IF bLoadTara THEN
	bLoadcell_fbcmd	:= LoadCell.GetTara();
END_IF
tmrLoadcellfbcmd(IN:= bLoadcell_fbcmd,PT:= T#2S);
IF tmrLoadcellfbcmd.Q THEN
	bLoadcell_fbcmd		:=FALSE;
	bLoadTara			:=FALSE;
	bLoadcell_Loadcail	:=FALSE;
	bLoadcell_Percent	:=FALSE;
	bLoadcell_RefLoad	:=FALSE;
	bLoadcell_MaxLoad	:=FALSE;
END_IF

ACTION Initial:
MC_GearIn(Master:= Axis_DualServo1,Slave:= Axis_DualServo2,Execute	:= FALSE);
MC_MoveVelocity(Axis:= Axis_DualServo1 ,Velocity := dualtestVelo,Execute:= FALSE);
MC_Stop(Axis := Axis_DualServo1,Execute:= FALSE);
tmrDelay(IN:=FALSE);
END_ACTION

ACTION TestDualServoCycleLeng:
IF Axis_DualServo1.Error OR Axis_DualServo2.Error THEN
	bDualRingCycleTest	:=FALSE;
	nStep:= 0;
END_IF


CASE nStep OF
	0:
		IF bDualRingCycleTest THEN
			Initial();
			nStep:= 5;
		END_IF
	5:

	
		IF Axis_DualServo1.ServoOn() AND Axis_DualServo2.ServoOn() THEN
			nStep:= 6;
		END_IF
	6:
		IF Axis_DualServo1.Status.StandStill AND Axis_DualServo2.Status.StandStill THEN
			nStep:= 7;
		END_IF
	7:
		MC_GearIn(Master:= Axis_DualServo1,Slave:= Axis_DualServo2,Execute	:= TRUE);
		IF 	MC_GearIn.InGear THEN
			nStep:= 10;
		END_IF
	10:
		MC_MoveVelocity(Axis:= Axis_DualServo1  ,Velocity := dualtestVelo);
	

		IF NOT bDualRingCycleTest THEN
			nStep:= 20;
		END_IF
		
	20:
		MC_Stop(Axis := Axis_DualServo1,Execute:= TRUE);
		IF MC_Stop.Done THEN
			nStep:= 25;
		END_IF
	25:
		MC_Stop(Axis := Axis_DualServo1,Execute:= FALSE);		
		nStep:= 0;
	
END_CASE
END_ACTION

ACTION TestLoadCycleLeng:

END_ACTION

END_PROGRAM

// ---- 01_POUs/MAIN.TcPOU
PROGRAM MAIN
VAR

	bInitial	:BOOL:= TRUE;;				//初始化
	ResetTrigger,AutoRunInitTrigger,PB_StartTrigger,IntiStartTrigger 	:R_TRIG;
	AutoRunDownTrigger,InitailDownTrigger	:F_TRIG;
	i	:INT;
END_VAR

//常態掃描  
RunParameter.strName	:= F_TrimRightSpace(RunParameter.strName);
Manual_POU();
IF PB_Stop OR PB_EMG OR OP.bStop_Sign THEN
	OP.xAutoRuning				:= FALSE;
	OP.xInitialRuning			:=FALSE;	
	OP.bInitialSign				:=FALSE;
	OP.xAutoMode				:=FALSE;
	RB_CS_SysIO.qENABLE			:= FALSE;
	RB_KR_SysIO.qMOVE_ENABLE	:= FALSE;
	
	MainControl.StopAllAxes();	
	MainControl.StopMotor();
	MainControl.StopAir();
END_IF
IF OP.bReset THEN
	MainControl.ErrorReset();
END_IF

(*---------------模式切換-------------------*)
IF OP.xAutoRuning OR OP.xAutoRuning THEN
	OP.bChangeMode	:=FALSE;
END_IF

IF OP.bChangeMode THEN
	OP.bChangeMode	:=FALSE;

	IF NOT OP.xAutoMode THEN
		EventLogger.eEventType	:= 1;
		EventLogger.strEventText	:= 'Mode : Auto ';
		EventLogger();
		OP.xAutoMode	:= TRUE;
		ELSE
		EventLogger.eEventType	:= 1;
		EventLogger.strEventText	:= 'Mode : Manual ';
		EventLogger();	
		OP.xAutoMode	:= FALSE;
	END_IF;
END_IF;
(*Stop*)



(*-------------POU Call ---------------*)
IF OP.xAutoRuning THEN
	OP.bInitialSign		:=FALSE;
END_IF;
IF NOT OP.xAutoMode THEN
	OP.xInitialDone	:=FALSE;
	OP.bStart		:=FALSE;
END_IF


PB_StartTrigger(CLK:=OP.bStart );
IntiStartTrigger(CLK:=OP.bInitialSign);
InitailDownTrigger(CLK:=OP.xInitialRuning);

IF OP.xAutoMode THEN
	IF IntiStartTrigger.Q THEN
		Initial_POU.FB_init(FALSE,FALSE);
		IF NOT OP.xAutoRuning THEN
			OP.xInitialRuning		:= TRUE;
			EventLogger.eEventType	:= 2;
			EventLogger.strEventText	:= 'Initial Runing ';
			EventLogger();
			ELSE
			EventLogger.eEventType	:= 4;
			EventLogger.strEventText	:= 'AutoRuning Do not Initial ';
			EventLogger();
		END_IF;
	END_IF;		
	IF PB_StartTrigger.Q AND NOT OP.xAutoRuning THEN
		IF NOT OP.xInitialRuning THEN
			OP.xAutoRuning	:= TRUE;
			EventLogger.eEventType	:= 2;
			EventLogger.strEventText	:= 'Auto Runing ';
			EventLogger();
			ELSE
			EventLogger.eEventType	:= 4;
			EventLogger.strEventText	:= 'Initial Runing,Please Waitting ';
			EventLogger();
		END_IF
	END_IF
END_IF

IF OP.xInitialRuning THEN
	Initial_POU();
END_IF
IF InitailDownTrigger.Q THEN
	MainControl.SoftStopAxis();
END_IF

IF OP.xAutoRuning THEN
	Automatic_POU();
END_IF

END_PROGRAM

// ---- 01_POUs/static/Manual_POU.TcPOU
PROGRAM Manual_POU
VAR
	fbGeneralAxis:ARRAY [1..6]OF FB_AxisGeneral;
	Clear							:ST_HMIAxieControl;
	HMIAxis_Box,HMIAxis_Dual1,HMIAxis_Dual2,HMIAxis_flyin,HMIAxis_load1,HMIAxis_load2				:ST_HMIAxieControl;
	wAxisNumb,wControlNumb,nChangeStep	:INT;
	tmrChangeMode			:TON;
	wTemp,i		:INT;
	bHMI_VerticalRoller , bHMI_VerticalBelt	:BOOL;
	bHMI_UnboxingInitial	,bHMI_UnboxingInitialDone,bHMI_UnboxingStart,bHMI_UnboxingDone:BOOL;
	bDualGearIn,bDualGearOut	:BOOL;
	MC_GearIn,MC_GearInload:MC_GearIn;
	MC_GearOut,MC_GearOutload:MC_GearOut;
	A1TouchPos,A2TouchPos					:ARRAY [1..5] OF LREAL;
	tempA1,tempA2	:LREAL;
	fbMC_UngroupAllAxes	: MC_UngroupAllAxes;
	fbMC_GroupDisable	: MC_GroupDisable;
	
END_VAR

Roller();
Axis();

ACTION Axis:
fbGeneralAxis[1](Axis:= Axis_FlyIn,HmiPanel:= HMIAxis_flyin);
fbGeneralAxis[2](Axis:= Axis_DualServo1,HmiPanel:= HMIAxis_Dual1);
fbGeneralAxis[3](Axis:= Axis_DualServo2,HmiPanel:= HMIAxis_Dual2);
fbGeneralAxis[4](Axis:= Axis_BoxPullOut,HmiPanel:= HMIAxis_Box,i_homecam:= NOT Sen_AxisBoxORG);	
fbGeneralAxis[5](Axis:= Axis_load1,HmiPanel:= HMIAxis_load1);
fbGeneralAxis[6](Axis:= Axis_load2,HmiPanel:= HMIAxis_load2);

MC_GearIn(
	Master:= Axis_DualServo1, 
	Slave:= Axis_DualServo2, 
	Execute:= bDualGearIn, 
	RatioNumerator:= , 
	RatioDenominator:= , 
	Acceleration:= , 
	Deceleration:= , 
	Jerk:= , 
	BufferMode:= , 
	Options:= , 
	InGear=> , 
	Busy=> , 
	Active=> , 
	CommandAborted=> , 
	Error=> , 
	ErrorID=> );

MC_GearOut(
	Slave:= Axis_DualServo2, 
	Execute:= bDualGearOut, 
);		

MC_GearInload(
	Master:= Axis_load1, 
	Slave:= Axis_load2, 
	Execute:= , 
	RatioNumerator:= , 
	RatioDenominator:= , 
	Acceleration:= , 
	Deceleration:= , 
	Jerk:= , 
	BufferMode:= , 
	Options:= , 
	InGear=> , 
	Busy=> , 
	Active=> , 
	CommandAborted=> , 
	Error=> , 
	ErrorID=> );

MC_GearOutload(
	Slave:= Axis_load2, 
	Execute:= , 
);		
UngroupAllAxes();
END_ACTION

ACTION Roller:
IF bHMI_VerticalRoller THEN
	AssRoller.Roller();	
END_IF

IF bHMI_VerticalBelt THEN
	AssRoller.Belt();	
END_IF
END_ACTION

ACTION Seizure:
(*
tmrChangeMode(PT:=T#1S);



CASE wControlNumb OF
	0:
		fbGeneralAxis[1](Axis:= Axis_FlyIn,HmiPanel:= HMIControlAxis);
	1:
		fbGeneralAxis[2](Axis:= Axis_Conv1,HmiPanel:= HMIControlAxis);
	2:
		fbGeneralAxis[3](Axis:= Axis_Conv2,HmiPanel:= HMIControlAxis);
	3:
		fbGeneralAxis[4](Axis:= Axis_BoxPullOut,HmiPanel:= HMIControlAxis);	
	4:
		fbGeneralAxis[5](Axis:= Axis_Unload1,HmiPanel:= HMIControlAxis);
	5:
		fbGeneralAxis[6](Axis:= Axis_Unload2,HmiPanel:= HMIControlAxis);
END_CASE
CASE nChangeStep OF
	0:
		IF wTemp<> wAxisNumb THEN
			nChangeStep	 := 5 ;
		END_IF; 

	5:
		HMIControlAxis:= Clear;
		tmrChangeMode(IN:= TRUE,PT:=T#1S);
		IF tmrChangeMode.Q THEN
			tmrChangeMode(IN:= FALSE);
			wControlNumb	:= wAxisNumb;
			nChangeStep	 	:= 0 ;
		END_IF


END_CASE


wTemp	:= wAxisNumb ;
*)
END_ACTION

METHOD UngroupAllAxes : BOOL
fbMC_GroupDisable(
	AxesGroup:= DualGroupRef, 
	Execute:= , 
	Done=> , 
	Busy=> , 
	Error=> , 
	ErrorId=> );	

fbMC_UngroupAllAxes(
	AxesGroup:= DualGroupRef, 
	Execute:= fbMC_GroupDisable.Done, 
	Done=> , 
	Busy=> , 
	Error=> , 
	ErrorId=> );	
	
UngroupAllAxes :=fbMC_UngroupAllAxes.Done AND fbMC_GroupDisable.Done;
END_METHOD

END_PROGRAM

// ---- 02_Unit/03_Axis/FB_AxisGeneral.TcPOU
FUNCTION_BLOCK FB_AxisGeneral
VAR_INPUT
	i_homecam		:BOOL;
	HmiPanel		:REFERENCE TO ST_HMIAxieControl;
	Axis 			:REFERENCE TO AXIS_REF_EXT;
END_VAR

VAR_OUTPUT
END_VAR

VAR
	fbReset: MC_Reset;
	fbJog: MC_Jog := (Mode := E_JOGMODE.MC_JOGMODE_CONTINOUS);

	fbStop: MC_Stop;
	fbMC_MoveAbsolute: MC_MoveAbsolute;
	fbMC_MoveRelative: MC_MoveRelative;
	fbMC_Home: MC_Home;
	strTemp	:WSTRING(50);
	ErrorTriger	:R_TRIG;
	nStep	:INT;
	tmrDef	:TON;
END_VAR

General_ACT();
StatusMapp();

CASE nStep OF
	0:
		IF HmiPanel.bServoSwitch THEN
			IF Axis.Status.StandStill THEN
				nStep	:=  10;
				ELSE	
				nStep	:=  5 ;
			END_IF
		END_IF
	5: //servo On
		IF Axis.ServoOn() THEN
			nStep	:=  20;
		END_IF
	10:
		IF Axis.ServoOFF() THEN
			nStep	:=  20;
		END_IF	
	20:
		HmiPanel.bServoSwitch	:= FALSE;
		nStep	:= 0;
END_CASE
//防呆跳回 
tmrDef(IN:= nStep <> 0 , PT:= T#1S);
IF tmrDef.Q THEN
	nStep	:= 20;
END_IF

ACTION General_ACT:
fbReset(
	Axis:=Axis , 
	Execute:= HmiPanel.bReset, 
	Done=> , 
	Busy=> , 
	Error=> , 
	ErrorID=> );
	
fbJog(
	Axis:= Axis , 
	JogForward:= HmiPanel.bJogF, 
	JogBackwards:=HmiPanel.bJogB , 
	Mode:= MC_JOGMODE_CONTINOUS, 
	Position:= , 
	Velocity:= HmiPanel.CommandVelo, 
	Acceleration:= , 
	Deceleration:= , 
	Jerk:= , 
	Done=> , 
	Busy=> , 
	Active=> , 
	CommandAborted=> , 
	Error=> , 
	ErrorID=> );	

fbStop(
	Axis:= Axis, 
	Execute:= HmiPanel.bSTOP , 
	Deceleration:= , 
	Jerk:= , 
	Options:= , 
	Done=> , 
	Busy=> , 
	Active=> , 
	CommandAborted=> , 
	Error=> , 
	ErrorID=> );

fbMC_MoveAbsolute(
	Axis:= AXIS, 
	Execute:= HmiPanel.bAbsPos, 
	Position:= HmiPanel.CommandAddres, 
	Velocity:= HmiPanel.CommandVelo, 
	Acceleration:= , 
	Deceleration:= , 
	Jerk:= , 
	BufferMode:= , 
	Options:= , 
	Done=> , 
	Busy=> , 
	Active=> , 
	CommandAborted=> , 
	Error=> , 
	ErrorID=> );
	
fbMC_MoveRelative(
	Axis:= Axis, 
	Execute:= HmiPanel.bINCPos, 
	Distance:= HmiPanel.CommandAddres, 
	Velocity:= HmiPanel.CommandVelo, 
	Acceleration:= , 
	Deceleration:= , 
	Jerk:= , 
	BufferMode:= , 
	Options:= , 
	Done=> , 
	Busy=> , 
	Active=> , 
	CommandAborted=> , 
	Error=> , 
	ErrorID=> );
	
fbMC_Home(
	Axis:=Axis , 
	Execute:=HmiPanel.bORG , 
	Position:= , 
	HomingMode:= , 
	BufferMode:= , 
	Options:= , 
	bCalibrationCam:=i_homecam , 
	Done=> , 
	Busy=> , 
	Active=> , 
	CommandAborted=> , 
	Error=> , 
	ErrorID=> );	


IF fbStop.Done THEN
	HmiPanel.bStop	:=FALSE;
END_IF
IF fbMC_MoveRelative.Done THEN
	HmiPanel.bINCPos	:=FALSE;
END_IF
IF fbMC_MoveAbsolute.Done THEN
	HmiPanel.CommandAddres	:= 0;
	HmiPanel.bAbsPos	:=FALSE;
END_IF
END_ACTION

ACTION StatusMapp:
	HmiPanel.moniDI						:= Axis.DI;
	HmiPanel.moniDeviceErrorCode		:= Axis.DeviceErrorcode;
	HmiPanel.bMoniReady					:= Axis.Status.StandStill;
	HmiPanel.bMoniDeviceError			:= Axis.Status.DriveDeviceError;
	HmiPanel.bMoniHomed					:= Axis.Status.Homed;
	HmiPanel.bMoniConpled				:= Axis.Status.Coupled;
	HmiPanel.bMoniControlLoopClosed		:= Axis.Status.ControlLoopClosed;
	HmiPanel.strStatus					:= Axis.strAxisStates;
END_ACTION

END_FUNCTION_BLOCK

// ---- 01_POUs/Initial_POU.TcPOU
PROGRAM Initial_POU
VAR
	nStep	:INT;
	strText	:STRING;
	aryBit	:ARRAY [0..100] OF BOOL;
	dwError: DWORD;
	tmrDelay,tmrDone	:TON;
END_VAR

CASE nStep OF
	0:
		tmrDelay(IN:=FALSE);
		tmrDone(IN:=FALSE);
		strText:= 'Intiail Runing';
		EventLogger.eEventType		:= 2;
		EventLogger.strEventText	:= 'Ini. Execute! ';	
		EventLogger();
		OP.xInitialDone				:=FALSE;
		nStep:= 5;
		IF LEN(RunParameter.strName) = 0 THEN
			nStep			:= 90;
			EventLogger.eEventType		:= 3;
			EventLogger.strEventText	:= 'Recipe Not Find ';	
			EventLogger();
			strText			:= 'Ini.Recipe Not Find';
		END_IF;
	5:
		tmrDelay(IN:=TRUE,PT:=T#5S);		
		IF tmrDelay.Q THEN
			strText:= 'Ini.Recipe Time Up ';
			EventLogger.eEventType		:= 3;
			EventLogger.strEventText	:= 'Recipe TimeUp ';	
			EventLogger();
			tmrDelay(IN:=FALSE);
			nStep			:= 90;
		END_IF	
			dwError:= RecipeManCommands.LoadAndWriteRecipe(RecipeDefinitionName:='Recipes' , RecipeName:=RunParameter.strName);	
			IF dwError = 0 THEN
				RunParameter	:= Edit_Parameter;
				strText:= 'Ini.Run Home ';
				nStep			:= 6;
				ELSE
				nStep			:= 90;
				strText:= 'Ini.Recipe Not Find';
				EventLogger.eEventType		:= 3;
				EventLogger.strEventText	:= 'Recipe Not Find ';	
				EventLogger();
			END_IF
	6:
		MainControl.ErrorReset();
		IF Air_Signal THEN
			nStep			:= 10;
			ELSE
			nStep			:= 90;
			strText:= 'Ini. Insuff. Air Pressure ';
			EventLogger.eEventType		:= 3;
			EventLogger.strEventText	:= ' Insuff. Air Pressure  ';	
			EventLogger();
		END_IF;		
	10:
		tmrDelay(IN:=TRUE,PT:=T#50S);		
		IF tmrDelay.Q THEN
			strText:= 'RB Init.TimeUp ';
			EventLogger.eEventType		:= 3;
			EventLogger.strEventText	:= ' RB Init.TimeUp ';	
			EventLogger();
			tmrDelay(IN:=FALSE);
			nStep			:= 90;
		END_IF	
	
		
		tmrDone(IN:= aryBit[7] AND aryBit[8],PT:=T#0.1S );
		aryBit[7]:=RB_CS.Initialization();
		aryBit[8]:=RB_KR.Initialization();					
		IF 	RB_CS.CommandError THEN
			strText:= 'RB Init. CS BOX Error ';
			EventLogger.eEventType		:= 3;
			EventLogger.strEventText	:= 'RB Init. CS BOX Error';	
			EventLogger();
			tmrDelay(IN:=FALSE);
			nStep			:= 90;
		END_IF
		IF tmrDone.Q THEN
			tmrDelay(IN:=FALSE);
			nStep	:= 20;	
		END_IF
	20:
		aryBit[0]:=M_DualServo.Initialization(FALSE);
		aryBit[1]:=M_Openbox1.Initialization(FALSE);
		aryBit[2]:=M_Sealing2.Initialization(FALSE);
		aryBit[3]:=M_LoadPic3.Initialization(FALSE);
		aryBit[4]:=M_UnloadNG4.Initialization(FALSE);
		aryBit[5]:=M_StackComv5.Initialization(FALSE);
		aryBit[6]:=M_RBStack6.Initialization(FALSE);
		tmrDelay(IN:=TRUE,PT:=T#50S);		
		IF tmrDelay.Q THEN
			strText:= 'Init. TimeUp ';
			EventLogger.eEventType		:= 3;
			EventLogger.strEventText	:= 'Hardware TimeUp';	
			EventLogger();
			tmrDelay(IN:=FALSE);
			nStep			:= 99;	
		END_IF
		tmrDone(IN:= aryBit[0] AND aryBit[1] AND aryBit[2] AND aryBit[3] AND aryBit[4] AND aryBit[5] AND aryBit[6] ,PT:=T#0.1S);
		IF  tmrDone.q THEN
			tmrDone(IN:=FALSE);
			tmrDelay(IN:=FALSE);
			EventLogger.eEventType		:= 1;
			EventLogger.strEventText	:= 'Intil. Complete';	
			EventLogger();
			strText:= 'Int.Finished';
			nStep			:= 50;
		END_IF;
		
	50:
		OP.xInitialDone	:= TRUE;	
	90:		
		EventLogger.eEventType		:= 3;
		EventLogger.strEventText	:= 'Ini. Cancel!';	
		EventLogger();	
		nStep			:= 91;	
END_CASE

METHOD FB_init : BOOL
VAR_INPUT
	bInitRetains : BOOL; // if TRUE, the retain variables are initialized (warm start / cold start)
	bInCopyCode : BOOL;  // if TRUE, the instance afterwards gets moved into the copy code (online change)
END_VAR
nStep	:= 0;
strText	:= '';
END_METHOD

END_PROGRAM

// ---- 01_POUs/Automatic_POU.TcPOU
PROGRAM Automatic_POU
VAR
	nStep 			:INT;
	bHlatMode,bNextStep		:BOOL;
END_VAR

//實例化

CASE  nStep OF
	0:
		M_Openbox1.Process(bHlatMode);
		M_Sealing2.Process(FALSE);
		M_LoadPic3.Process(FALSE);
		M_UnloadNG4.Process(FALSE);
		M_DualServo.Process(FALSE);
		M_StackComv5.Process(FALSE);
		M_RBStack6.Process(FALSE);
END_CASE
IF bNextStep THEN
	M_Openbox1.HaltStepContiune();
	bNextStep:=FALSE;
END_IF

END_PROGRAM

// ---- 01_POUs/static/UPS_POU.TcPOU
PROGRAM UPS_POU
VAR
	fbS_UPS_BAPI:FB_S_UPS_BAPI;
	bPowerFailDetect  : BOOL; (* TRUE while powerfailure is detected *)
    eState            : E_S_UPS_State; (* current ups state *)
    nCapacity         : BYTE; (* actual capacity of UPS *)
    bBusy             : BOOL; (* TRUE: function block is busy *)
    bError            : BOOL; (* FALSE: function block has error *)
    nErrID            : UDINT; (* FB error ID *)
END_VAR

fbS_UPS_BAPI(
	sNetID:= '', 
	iPLCPort:= 851, 
	tTimeout:= DEFAULT_ADS_TIMEOUT, 
	eUpsMode:= eSUPS_WrPersistData_Shutdown, 
	ePersistentMode:= SPDM_2PASS , 
	tRecoverTime:= T#10S, 
	bPowerFailDetect=> bPowerFailDetect, 
	eState=> eState, 
	nCapacity=> nCapacity, 
	bBusy=> bBusy, 
	bError=> bError, 
	nErrID=> nErrID);

END_PROGRAM

// ---- 02_Unit/01_Customization/Ass_Pallet.TcPOU
FUNCTION_BLOCK Ass_Pallet
VAR_INPUT
END_VAR
VAR_OUTPUT
END_VAR
VAR
END_VAR

END_FUNCTION_BLOCK

// ---- 02_Unit/99_Other/FB_RecordValue.TcPOU
FUNCTION_BLOCK FB_RecordValue
VAR_INPUT
END_VAR
VAR_OUTPUT
END_VAR
VAR
END_VAR

END_FUNCTION_BLOCK

// ---- 02_Unit/03_Axis/FB_ORG_PositiveEndLessByTouchprobe.TcPOU
FUNCTION_BLOCK FB_ORG_PositiveEndLessByTouchprobe
VAR_INPUT
	Axis		:AXIS_REF;
	Execute		:BOOL;
	Position	:LREAL;
	Velocity	:LREAL;
END_VAR
VAR_OUTPUT
	Error	:BOOL;
	Busy	:BOOL;
	Done	:BOOL;
END_VAR
VAR
	nStep	:INT;
	fbTrig	:R_TRIG;
	fbMC_MoveVelocity: MC_MoveVelocity;
	MC_TouchProbe: MC_TouchProbe;
	MC_AbortTrigger: MC_AbortTrigger;
	TRIGGER_REF	:TRIGGER_REF ;
	MC_ReadDriveAddress: MC_ReadDriveAddress;
	MC_Stop: MC_Stop;
	MC_Home: MC_Home;
	MC_SetPosition: MC_SetPosition;
END_VAR

fbTrig(CLK:=Execute);
Axis.ReadStatus();

IF fbTrig.Q THEN

	IF Axis.Status.StandStill THEN
		MC_ReadDriveAddress(Axis:= Axis,Execute:=FALSE);
		nStep	:=1;
	ELSE
		nStep	:= 99;
	END_IF;	
END_IF
		
CASE nStep OF
	1:		
		Busy:= TRUE;
		MC_ReadDriveAddress(
			Axis:= Axis, 
			Execute:=TRUE , 
			Done=> , 
			Busy=> , 
			Error=> , 
			ErrorID=> , 
			DriveAddress=> );
	IF MC_ReadDriveAddress.Done THEN
		Intial();
		nStep	:= 5;
	END_IF
5:
			MC_TouchProbe(
				Axis:= Axis, 
				TriggerInput:=TRIGGER_REF , 
				Execute:= TRUE, 
				WindowOnly:= , 
				FirstPosition:= , 
				LastPosition:= , 
				Done=> , 
				Busy=> , 
				CommandAborted=> , 
				Error=> , 
				ErrorID=> , 
				RecordedPosition=> , 
				RecordedData=> );	
			fbMC_MoveVelocity(
				Axis:= Axis, 
				Execute:= MC_TouchProbe.Busy, 
				Velocity:= Velocity, 
				Acceleration:= , 
				Deceleration:= , 
				Jerk:= , 
				Direction:= , 
				BufferMode:= , 
				Options:= , 
				InVelocity=> , 
				Busy=> , 
				Active=> , 
				CommandAborted=> , 
				Error=> , 
				ErrorID=> );	
		
			MC_Stop(
				Axis:= Axis, 
				Execute:=MC_TouchProbe.Done , 
				Deceleration:= , 
				Jerk:= , 
				Options:= , 
				Done=> , 
				Busy=> , 
				Active=> , 
				CommandAborted=> , 
				Error=> , 
				ErrorID=> );
			IF Axis.Status.MotionState = MC_AXISSTATE_STOPPING THEN	
				nStep	:= 10;
				END_IF;
10:	
	IF Axis.Status.MotionState = MC_AXISSTATE_STANDSTILL THEN
		nStep	:= 15;
	END_IF
			MC_Stop(
				Axis:= Axis, 
				Execute:= FALSE, 
				Deceleration:= , 
				Jerk:= , 
				Options:= , 
				Done=> , 
				Busy=> , 
				Active=> , 
				CommandAborted=> , 
				Error=> , 
				ErrorID=> );
	15:
		MC_SetPosition(
		Axis:= Axis, 
		Execute:= TRUE, 
		Position:=Axis.NcToPlc.ActPos - MC_TouchProbe.RecordedPosition ,
		Mode:= , 
		Options:= , 
		Done=> , 
		Busy=> , 
		Error=> , 
		ErrorID=> );
	IF MC_SetPosition.Done	THEN
		MC_Home.Execute:=TRUE;
	END_IF
	MC_Home(
		Axis:= Axis, 
		Execute:= , 
		Position:=(Axis.NcToPlc.ActPos - MC_TouchProbe.RecordedPosition) - Position, 
		HomingMode:= MC_ForceCalibration, 
		BufferMode:= , 
		Options:= , 
		bCalibrationCam:= , 
		Done=> , 
		Busy=> , 
		Active=> , 
		CommandAborted=> , 
		Error=> , 
		ErrorID=> );
	IF MC_Home.Done	THEN
		nStep:=20;
	END_IF
	20:
	Busy	:=FALSE;
	Done	:=TRUE;		
	IF NOT Execute THEN
		Done	:=FALSE;		
		nStep	:= 0;
	END_IF
END_CASE

METHOD FB_init : BOOL
VAR_INPUT
	bInitRetains : BOOL; // if TRUE, the retain variables are initialized (warm start / cold start)
	bInCopyCode : BOOL;  // if TRUE, the instance afterwards gets moved into the copy code (online change)
END_VAR
END_METHOD

METHOD INTERNAL Intial : BOOL
VAR_INPUT
END_VAR
TRIGGER_REF.EncoderID			:= Axis.DriveAddress.NcAxisId;
TRIGGER_REF.TouchProbe			:= Tc2_MC2.TouchProbe1;
TRIGGER_REF.SignalSource		:= Tc2_MC2.SignalSource_Default;
TRIGGER_REF.Mode				:= Tc2_MC2.TOUCHPROBEMODE_SINGLE;

	fbMC_MoveVelocity(Axis:= Axis, Execute:= FALSE);
	MC_TouchProbe(Axis:= Axis,TriggerInput:=TRIGGER_REF ,Execute:= FALSE);
	MC_AbortTrigger(Axis:= Axis,TriggerInput:=TRIGGER_REF ,Execute:= FALSE);
	MC_ReadDriveAddress(Axis:= Axis, Execute:= FALSE);
	MC_Stop(Axis:= Axis, Execute:= FALSE);
	MC_Home(Axis:= Axis, Execute:= FALSE);
	MC_SetPosition(Axis:= Axis, Execute:= FALSE);
END_METHOD

END_FUNCTION_BLOCK

// ---- GlobalTextList.TcGTLO
TEXTLIST GlobalTextList
  229 = '%4.1f'
  568 = '%6.2f'
  145 = '%8.1f'
  917 = '%b'
  32 = '%d'
  787 = '%f'
  907 = '%s'
  823 = 'Coil'
  994 = 'Conve Loadin'
  45 = 'Conve ORG'
  1009 = 'Coupled'
  815 = 'Duel'
  812 = 'GearInPosition'
  37 = 'Group'
  1006 = 'HasJob'
  1007 = 'Homed'
  333 = 'Ini'
  1008 = 'InPosit'
  397 = 'LatchPosition'
  345 = 'LEFT'
  404 = 'Left ORG'
  643 = 'LoadIn'
  752 = 'Modechg'
  836 = 'Moving'
  1004 = 'PackingComvAxis'
  242 = 'POU_Comv.bStDuel'
  999 = 'Power'
  241 = 'Remove'
  768 = 'Reset'
  595 = 'ResIn'
  365 = 'Right'
  678 = 'Right ORG'
  998 = 'Run'
  962 = 'ScanIn'
  44 = 'slot[INDEX].GearInPosition'
  43 = 'slot[INDEX].LatchPosition'
  921 = 'Start'
  93 = 'Step %s'
  6 = 'Test'
  506 = 'WriteIn'
  1000 = '位置 : %2.2f mm'
  741 = '入料'
  711 = '入料位置'
  255 = '入料格數'
  256 = '入料點'
  642 = '出料位置'
  358 = '出料點'
  400 = '前輸送引入距離'
  624 = '前輸送速度'
  961 = '數量%s'
  1001 = '現在位置'
  700 = '輸送帶_模組長度'
  948 = '輸送帶_每隔長度'
  140 = '輸送帶_膜長度'
  274 = '輸送帶引入距離'
  152 = '輸送帶總長'
  939 = '輸送帶速度'
  1003 = '速度'
  1002 = '速度 : %2.2f mm/s'
  751 = '雙伺服安全距離'
END_TEXTLIST
